FUNCTION_BLOCK FB_ExternalSetpointGenerator IMPLEMENTS I_ExternalSetpointGenerator
VAR CONSTANT
    nOFFSET_TO_NCTOPLC_AXIS_REF_STATE : LWORD := 0;
END_VAR
VAR
    iMotionAxis : I_MotionAxis;

    AxisReference : REFERENCE TO AXIS_REF;

    AxisReference_NcToPlc_StateDWord : NCTOPLC_AXIS_REF_STATE;

    bEnableCommanded : BOOL;
    fbEnableSetPointGenerator : MC_ExtSetPointGenEnable;

    bDisableCommanded : BOOL;
    fbDisableSetPointGenerator : MC_ExtSetPointGenDisable;

    bHaltCommanded : BOOL;
    fbHalt : MC_Halt;

    bEnableBusy : BOOL;
    bEnableDone : BOOL;
END_VAR


AxisReference REF= iMotionAxis.GetAxisRef();

MEMCPY(
    ADR(AxisReference_NcToPlc_StateDWord),
    ADR(AxisReference.NcToPlc) + nOFFSET_TO_NCTOPLC_AXIS_REF_STATE,
    SIZEOF(AxisReference_NcToPlc_StateDWord)
);

fbEnableSetPointGenerator(
    Axis := THIS^.AxisReference,
    Execute := bEnableCommanded
);
bEnableCommanded := FALSE;

fbDisableSetPointGenerator(
    Axis := THIS^.AxisReference,
    Execute := bDisableCommanded
);
bDisableCommanded := FALSE;

fbHalt(
    Axis := THIS^.AxisReference,
    Execute := bHaltCommanded
);
bHaltCommanded := FALSE;


METHOD PUBLIC Disable
VAR_OUTPUT
    Done : BOOL;
    Busy : BOOL;
    Error : BOOL;
    ErrorID : UDINT;
    Enabled : BOOL;
END_VAR

bDisableCommanded := TRUE;

fbDisableSetPointGenerator(
    Axis := THIS^.AxisReference,
    Done => Done,
    Busy => Busy,
    Error => Error,
    ErrorID => ErrorID,
    Enabled => Enabled
);
END_METHOD


PROPERTY DisableBusy : BOOL
GET

DisableBusy := fbDisableSetPointGenerator.Busy;
END_GET
END_PROPERTY


PROPERTY DisableDone : BOOL
GET

DisableDone := fbDisableSetPointGenerator.Done;
END_GET
END_PROPERTY


METHOD PUBLIC Enable
VAR_OUTPUT
    Done : BOOL;
    Busy : BOOL;
    Error : BOOL;
    ErrorID : UDINT;
    Enabled : BOOL;
END_VAR

IF iMotionAxis.PowerIsEnabled AND iMotionAxis.PositiveMotionIsEnabled AND iMotionAxis.NegativeMotionIsEnabled THEN
    bEnableCommanded := TRUE;
END_IF

fbEnableSetPointGenerator(
    Axis := THIS^.AxisReference,
    PositionType := E_PositionType.POSITIONTYPE_ABSOLUTE,
    Done => bEnableDone,
    Busy => bEnableBusy,
    Error => Error,
    ErrorID => ErrorID,
    Enabled => Enabled
);
END_METHOD


PROPERTY EnableBusy : BOOL
GET

EnableBusy := fbEnableSetPointGenerator.Busy;
END_GET
END_PROPERTY


PROPERTY EnableDone : BOOL
GET

EnableDone := fbEnableSetPointGenerator.Done;
END_GET
END_PROPERTY


PROPERTY EnableError : BOOL
GET

EnableError := fbEnableSetPointGenerator.Error;
END_GET
END_PROPERTY


METHOD FB_Init: BOOL
VAR_INPUT
    bInitRetains: BOOL; // TRUE: the retain variables are initialized (reset warm / reset cold)
    bInCopyCode: BOOL;  // TRUE: the instance will be copied to the copy code afterward (online change)

    iMotionAxis : I_MotionAxis;
END_VAR

THIS^.iMotionAxis := iMotionAxis;
END_METHOD


METHOD PUBLIC Halt
VAR_OUTPUT
    Done : BOOL;
    Busy : BOOL;
    Active : BOOL;
    CommandAborted : BOOL;
    Error : BOOL;
    ErrorID : UDINT;
END_VAR

fbHalt(
    Axis := THIS^.AxisReference,
    Execute := TRUE,
    Done => Done,
    Busy => Busy,
    Active => Active,
    CommandAborted => CommandAborted,
    Error => Error,
    ErrorID => ErrorID
);
END_METHOD

PROPERTY HaltBusy : BOOL
GET

HaltBusy := fbHalt.Busy;
END_GET
END_PROPERTY

PROPERTY HaltDone : BOOL
GET

HaltDone := fbHalt.Done;
END_GET
END_PROPERTY


METHOD PUBLIC IsEnabled : BOOL

IsEnabled := AxisReference_NcToPlc_StateDWord.14 AND fbEnableSetPointGenerator.Enabled;
END_METHOD


METHOD PUBLIC SetAcceleraSetpoint
VAR_INPUT
    Setpoint : LREAL;
END_VAR
VAR_OUTPUT
    Error : BOOL;
    ErrorMsg : T_MaxString;
END_VAR

SetSetpoints(
    PositionSetpoint := THIS^.AxisReference.NcToPlc.SetPos,
    VelocitySetpoint := THIS^.AxisReference.NcToPlc.SetVelo,
    AcceleraSetpoint := Setpoint,
    Error => Error,
    ErrorMsg => ErrorMsg
);
END_METHOD


METHOD PUBLIC SetPositionSetpoint
VAR_INPUT
    Setpoint : LREAL;
END_VAR
VAR_OUTPUT
    Error : BOOL;
    ErrorMsg : T_MaxString;
END_VAR

SetSetpoints(
    PositionSetpoint := Setpoint,
    VelocitySetpoint := THIS^.AxisReference.NcToPlc.SetVelo,
    AcceleraSetpoint := THIS^.AxisReference.NcToPlc.SetAcc,
    Error => Error,
    ErrorMsg => ErrorMsg
);
END_METHOD


METHOD PUBLIC SetSetpoints
VAR_INPUT
    PositionSetpoint : LREAL;
    VelocitySetpoint : LREAL;
    AcceleraSetpoint : LREAL;
END_VAR
VAR_OUTPUT
    Error : BOOL;
    ErrorMsg : T_MaxString;
END_VAR
VAR
    nDirection : DINT;
END_VAR

IF NOT THIS^.iMotionAxis.PowerIsEnabled THEN
    Error := TRUE;
    ErrorMsg := 'Cannot set external setpoint due to axis power being disabled.';
    RETURN;
END_IF

IF PositionSetpoint < THIS^.AxisReference.NcToPlc.ActPos THEN
    nDirection := -1;
ELSE
    nDirection := 1;
END_IF

IF nDirection = 1 AND NOT THIS^.iMotionAxis.PositiveMotionIsEnabled THEN
    Error := TRUE;
    ErrorMsg := 'Cannot set setpoint in the positive direction because positive motion is disabled.';
    RETURN;
END_IF

IF nDirection = -1 AND NOT THIS^.iMotionAxis.NegativeMotionIsEnabled THEN
    Error := TRUE;
    ErrorMsg := 'Cannot set setpoint in the negative direction because negative motion is disabled.';
    RETURN;
END_IF

MC_ExtSetPointGenFeed(
    Position := PositionSetpoint,
    Velocity := VelocitySetpoint,
    Acceleration := AcceleraSetpoint,
    Direction := nDirection,
    Axis := THIS^.AxisReference
);
END_METHOD


METHOD PUBLIC SetVelocitySetpoint
VAR_INPUT
    Setpoint : LREAL;
END_VAR
VAR_OUTPUT
    Error : BOOL;
    ErrorMsg : T_MaxString;
END_VAR

SetSetpoints(
    PositionSetpoint := THIS^.AxisReference.NcToPlc.SetPos,
    VelocitySetpoint := Setpoint,
    AcceleraSetpoint := THIS^.AxisReference.NcToPlc.SetAcc,
    Error => Error,
    ErrorMsg => ErrorMsg
);
END_METHOD

END_FUNCTION_BLOCK

(* stored: Version 1.1.0.1, ProductVersion 3.1.4026.11
   POU FB_ExternalSetpointGenerator: Id {48348351-f54a-4182-b51d-178baa336e3e}, SpecialFunc None
   Method Disable: Id {2405d3c1-712a-4c9d-8b0e-e64f64d46922}
   Property DisableBusy: Id {ebc0196e-70f0-4ec8-8965-7bf2af41f9a7}
   Get Get: Id {3c34d3c2-fdc1-4919-924d-806fc91e5052}
   Property DisableDone: Id {3ede6098-89b4-4dc5-b10f-3f70168e307e}
   Get Get: Id {ac9144d6-7b29-46a3-b5ef-645b7d85779a}
   Method Enable: Id {248900d9-87ae-4693-b478-0b8aa22cc50b}
   Property EnableBusy: Id {6da14380-8aec-44a0-b296-4971e0590319}
   Get Get: Id {fafba1ec-aa62-4816-9164-d0e808545724}
   Property EnableDone: Id {fe053b89-d979-4f23-9180-6fbada24cb77}
   Get Get: Id {8e61fe3c-7012-45e5-b873-8425f2cbec64}
   Property EnableError: Id {aa38d092-dd85-4db1-8c2f-5f772a359ac6}
   Get Get: Id {1d8a418c-a427-43b4-a6b4-02816c244598}
   Method FB_Init: Id {9fdaf2df-47d9-4baa-b3d4-f388e1f1371d}
   Method Halt: Id {f67e4245-e771-4009-9436-72c09ac49ef1}
   Property HaltBusy: Id {db5ca45d-5fc4-41e8-97b2-88d044c7038b}
   Get Get: Id {211a40b7-0841-43b1-9620-818cf3495485}
   Property HaltDone: Id {c1a8896b-673b-4892-91bf-6ca1ffd898c9}
   Get Get: Id {a21d75a9-7a11-4932-96fe-33576c98315b}
   Method IsEnabled: Id {d118f580-9ab1-4d2f-8e49-7eb2fcd933d6}
   Method SetAcceleraSetpoint: Id {35f50744-9fb8-4c6b-bc0e-8091dd561e37}
   Method SetPositionSetpoint: Id {d2ea1ddb-aefd-4201-8f1e-056bbb7a842a}
   Method SetSetpoints: Id {f7c477cb-0de8-404f-a125-ae3823ead4c2}
   Method SetVelocitySetpoint: Id {8151fa4c-3612-4a0c-89e6-e25694690391} *)
